# EPICS substitutions: iocBoot/iocvirPV/DPU06.substitutions
file "../../db/virAi.template"{ pattern
{DPU,    num,    Temp}
{06,    0,    500}
{06,    1,    500}
{06,    2,    500}
{06,    3,    500}
{06,    4,    500}
{06,    5,    500}
{06,    6,    500}
{06,    7,    500}
{06,    8,    500}
{06,    9,    500}
{06,    10,    500}
{06,    11,    500}
{06,    12,    500}
{06,    13,    500}
{06,    14,    500}
{06,    15,    500}
{06,    16,    500}
{06,    17,    500}
{06,    18,    500}
{06,    19,    500}
{06,    20,    500}
{06,    21,    500}
{06,    22,    500}
{06,    23,    500}
{06,    24,    500}
{06,    25,    500}
{06,    26,    500}
{06,    27,    500}
{06,    28,    500}
{06,    29,    500}
{06,    30,    500}
{06,    31,    500}
{06,    32,    500}
{06,    33,    500}
{06,    34,    500}
{06,    35,    500}
{06,    36,    500}
{06,    37,    500}
{06,    38,    500}
{06,    39,    500}
{06,    40,    500}
{06,    41,    500}
{06,    42,    500}
{06,    43,    500}
{06,    44,    500}
{06,    45,    500}
{06,    46,    500}
{06,    47,    500}
{06,    48,    500}
{06,    49,    500}
{06,    50,    500}
{06,    51,    500}
{06,    52,    500}
{06,    53,    500}
{06,    54,    500}
{06,    55,    500}
{06,    56,    500}
{06,    57,    500}
{06,    58,    500}
{06,    59,    500}
{06,    60,    500}
{06,    61,    500}
{06,    62,    500}
{06,    63,    500}
{06,    64,    500}
{06,    65,    500}
{06,    66,    500}
{06,    67,    500}
{06,    68,    500}
{06,    69,    500}
{06,    70,    500}
{06,    71,    500}
{06,    72,    500}
{06,    73,    500}
{06,    74,    500}
{06,    75,    500}
{06,    76,    500}
{06,    77,    500}
{06,    78,    500}
{06,    79,    500}
{06,    80,    500}
{06,    81,    500}
{06,    82,    500}
{06,    83,    500}
{06,    84,    500}
{06,    85,    500}
{06,    86,    500}
{06,    87,    500}
{06,    88,    500}
{06,    89,    500}
{06,    90,    500}
{06,    91,    500}
{06,    92,    500}
{06,    93,    500}
{06,    94,    500}
{06,    95,    500}
{06,    96,    500}
{06,    97,    500}
{06,    98,    500}
{06,    99,    500}
{06,    100,    500}
{06,    101,    500}
{06,    102,    500}
{06,    103,    500}
{06,    104,    500}
{06,    105,    500}
{06,    106,    500}
{06,    107,    500}
{06,    108,    500}
{06,    109,    500}
{06,    110,    500}
{06,    111,    500}
{06,    112,    500}
{06,    113,    500}
{06,    114,    500}
{06,    115,    500}
{06,    116,    500}
{06,    117,    500}
{06,    118,    500}
{06,    119,    500}
{06,    120,    500}
{06,    121,    500}
{06,    122,    500}
{06,    123,    500}
{06,    124,    500}
{06,    125,    500}
{06,    126,    500}
{06,    127,    500}
{06,    128,    500}
{06,    129,    500}
{06,    130,    500}
{06,    131,    500}
{06,    132,    500}
{06,    133,    500}
{06,    134,    500}
{06,    135,    500}
{06,    136,    500}
{06,    137,    500}
{06,    138,    500}
{06,    139,    500}
{06,    140,    500}
{06,    141,    500}
{06,    142,    500}
{06,    143,    500}
{06,    144,    500}
{06,    145,    500}
{06,    146,    500}
{06,    147,    500}
{06,    148,    500}
{06,    149,    500}
{06,    150,    500}
{06,    151,    500}
{06,    152,    500}
{06,    153,    500}
{06,    154,    500}
{06,    155,    500}
{06,    156,    500}
{06,    157,    500}
{06,    158,    500}
{06,    159,    500}
{06,    160,    500}
{06,    161,    500}
{06,    162,    500}
{06,    163,    500}
{06,    164,    500}
{06,    165,    500}
{06,    166,    500}
{06,    167,    500}
{06,    168,    500}
{06,    169,    500}
{06,    170,    500}
{06,    171,    500}
{06,    172,    500}
{06,    173,    500}
{06,    174,    500}
{06,    175,    500}
{06,    176,    500}
{06,    177,    500}
{06,    178,    500}
{06,    179,    500}
{06,    180,    500}
{06,    181,    500}
{06,    182,    500}
{06,    183,    500}
{06,    184,    500}
{06,    185,    500}
{06,    186,    500}
{06,    187,    500}
{06,    188,    500}
{06,    189,    500}
{06,    190,    500}
{06,    191,    500}
{06,    192,    500}
{06,    193,    500}
{06,    194,    500}
{06,    195,    500}
{06,    196,    500}
{06,    197,    500}
{06,    198,    500}
{06,    199,    500}
}
